PROGRAM MAIN
VAR
	fbRemoteControl : PalletizerRemoteCtrl;
	fbPalletizer : Palletizer;
END_VAR

fbPalletizer();
fbRemoteControl(fbPalletizer := fbPalletizer);

END_PROGRAM

(* stored: Version 1.1.0.1, ProductVersion 3.1.4024.2
   POU MAIN: Id {7295c37b-1171-4097-8fbe-9dd92cbb79f6}, SpecialFunc None *)
